{attribute 'hide_all_locals'}
FUNCTION_BLOCK PUBLIC FB_ContractEmployee_2 EXTENDS FB_Employee_1
VAR_INPUT
END_VAR
VAR_OUTPUT
END_VAR
VAR
	nHourlyPayBacking		:	UINT;
	nMonthlyHoursBacking	:	UINT;
END_VAR

METHOD PUBLIC GetMonthlySalary : LREAL
VAR_INPUT
END_VAR
GetMonthlySalary := nMonthlyHours * nHourlyPay;
END_METHOD

{attribute 'monitoring' := 'variable'}
PROPERTY PUBLIC nHourlyPay : UINT
GET
nHourlyPay := nHourlyPayBacking;
END_GET
SET
nHourlyPayBacking := nHourlyPay;
END_SET
END_PROPERTY

{attribute 'monitoring' := 'variable'}
PROPERTY PUBLIC nMonthlyHours : UINT
GET
nMonthlyHours := nMonthlyHoursBacking;
END_GET
SET
nMonthlyHoursBacking := nMonthlyHours;
END_SET
END_PROPERTY

END_FUNCTION_BLOCK

(* stored: Version 1.1.0.1, ProductVersion 3.1.4024.12
   POU FB_ContractEmployee_2: Id {c95723a0-cc2b-4163-ac14-a3ce520e2a04}, SpecialFunc None
   Method GetMonthlySalary: Id {b476780b-bf60-4517-a27d-10f90bbbfefd}
   Property nHourlyPay: Id {f92853b4-68b5-48f0-804c-56be801a470f}
   Get Get: Id {c566c18c-1dca-4565-bee7-f47cc650fe47}
   Set Set: Id {899ca572-f74e-43b8-9a9e-1c911edee194}
   Property nMonthlyHours: Id {2fdc0080-170a-42f1-8a6b-44630117664a}
   Get Get: Id {65306d45-cbf4-4435-8653-c51df6bc280d}
   Set Set: Id {e354902e-0201-448c-a8d1-3b3b6b839fd5} *)
